// TIA Portal V19 export
VAR_GLOBAL   // PLC tag table "U2Em5_Input"
   inspectionAfterPlasticTrayJackingU2EM5 AT %I47.1 : Bool;   // U2EM5_ Plastic Jacking Post Detection / Em120_塑胶顶升后检测
   plasticTrayTrayInplaceDetectionU2EM5 AT %I46.5 : Bool;   // U2EM5_ Plastic tray in place detection / Em120_塑胶托盘到位检测
   plasticTrayLiftingCylinderworkingPositionDetectionU2EM5_1 AT %I46.6 : Bool;   // U2EM5-Plastic Jacking Cylinder 1 Working Position Detection / Em120_塑胶顶升气缸1工作位检测
   plasticTrayFeedingDetectionU2EM5 AT %I46.4 : Bool;   // U2EM5_ Plastic tray feeding detection / Em120_塑胶托盘入料检测
   inspectionBeforePlasticTrayJackingU2EM5 AT %I47.0 : Bool;   // U2EM5_Plastic Jacking Pre Inspection / Em120_塑胶顶升前检测
   plasticTrayLiftingCylinderHomePositionDetectionU2EM5_1 AT %I46.7 : Bool;   // U2EM5-Plastic Jacking Cylinder 1 in situ Detection / Em120_塑胶顶升气缸1原位检测
   scapegoat1SignalU2EM5 AT %I47.2 : Bool;   // Em120_替罪羊1信号
   scapegoat2SignalU2EM5 AT %I47.3 : Bool;   // Em120_替罪羊2信号
END_VAR
